DATA_BLOCK "FF_IO"
{ S7_Optimized_Access := 'FALSE' }
VERSION : 0.1
NON_RETAIN
   VAR
      FanSpeed : Real;        // fan.speed (PLC writes) airflow reference, 0..100 %; the fan ramps towards it
      OvenHeater : Real;      // oven.heater (PLC writes) heater power, 0..100 %
      TempGaugeValue : Real;  // temp_gauge.value (PLC writes) needle position, scale 0..250 C
      FanRun : Bool;          // fan.run (PLC writes) run the fan
      PanelGreen : Bool;      // panel.green (PLC writes) green lamp on the panel
      PanelRed : Bool;        // panel.red (PLC writes) red lamp on the panel
      TowerGreen : Bool;      // tower.green (PLC writes) tower lamp, green
      TowerRed : Bool;        // tower.red (PLC writes) tower lamp, red
      TowerYellow : Bool;     // tower.yellow (PLC writes) tower lamp, yellow
      FanAirflow : Real;      // fan.airflow (PLC reads) airflow actually delivered, % -- lags the reference, and reads 0 with the motor failed
      OvenTemperature : Real; // oven.temperature (PLC reads) plate temperature, degC
      PanelSetpoint : Real;   // panel.setpoint (PLC reads) the operator's pot, 40..200 C (starts at 150)
      FanFault : Bool;        // fan.fault (PLC reads) fan motor failed: TRUE = it takes your reference and blows nothing
      OvenAttemp : Bool;      // oven.attemp (PLC reads) within +/-3 degC of the station's own 150 degC -- not the pot
      OvenFault : Bool;       // oven.fault (PLC reads) element failed: TRUE = it takes your command and heats nothing
      PanelEstop : Bool;      // panel.estop (PLC reads) E-stop, normally closed: TRUE = healthy, FALSE = pressed; stays pressed until pulled out
      PanelReset : Bool;      // panel.reset (PLC reads) Reset button, momentary: a short pulse per press
      PanelStart : Bool;      // panel.start (PLC reads) Start button, momentary: a short pulse per press -- latch it
      PanelStop : Bool;       // panel.stop (PLC reads) Stop button, momentary: a short pulse per press
   END_VAR


BEGIN

END_DATA_BLOCK


FUNCTION_BLOCK "CoolingTunnel"
{ S7_Optimized_Access := 'TRUE' }
VERSION : 0.1

// ---------------------------------------------------------------------------
// FactoryForge starter -- Cooling tunnel (scene cooling-tunnel)
// Generated by tools/gen_starters.py; see README.md beside this file.
//
// THE TASK
//   Hold the product at the temperature on the panel's pot. The heater can
//   only push the temperature up and the room takes heat away slowly, so
//   the fan is how it comes down fast: split one controller's output,
//   heater above zero and fan below it, with a deadband between them.
//   Never run both at once. fan.speed is a reference -- the fan ramps, and
//   fan.airflow is what it is really delivering.
//
// DONE WHEN
//   The product settles within a few degrees of the pot and holds there.
//   Drop the pot 60 C and it comes down in seconds with the fan, not in a
//   quarter of a minute on the room; raise it again and the heater takes
//   back over with the fan stopped. A fan left running while the heater
//   trims holds every setpoint and heats the air it blows away -- watch
//   oven.heater and fan.airflow and they are never both up. Fail the fan
//   (fan.fault) and fan.speed keeps reading your reference while the
//   airflow collapses. The mushroom (panel.estop, normally closed) stops
//   the heater and the fan within 200 ms and its trip latches: releasing
//   it restarts nothing, and neither does Start or Reset alone -- only
//   Reset, then Start.
//
// Every signal is a member of the global DB "FF_IO" above: read and write
// them as "FF_IO".<Name>, e.g. "FF_IO".FanSpeed. Its comments say which
// way each one runs. Call this block from OB1 (drag it into Main; TIA creates
// the instance DB).
// ---------------------------------------------------------------------------

BEGIN

    // Your program.

END_FUNCTION_BLOCK
